(* Logix 5000 project; controller cal1615 1756-L62 rev 20.11; software revision 20.05; part 54 of 81 *)
(* tags used below, declared in another part *)
   FAULT : BOOL;   // Fault AFI
   p01_recipe_active : recipe;   // Active Recipe
   p01r09 : routine;   // System Modes
   p01r09_pb_global_reset : BOOL;   // System Modes PB: Global Fault Reset
   p01r13_line_running : BOOL;   // System Line Start Sequence Line Running
   p02_dint_from_hmi : hmi_dint;
   p02_real_from_hmi : hmi_real;   // MOP HMI Iface Real from HMI
   p23_ao_servo_ds_jog_vel_cmd : REAL;   // Impreg Servo Drive Side Jog Velocity Command [in/sec]
   p23_ao_servo_ds_position_cmd : REAL;   // Impreg Servo Drive Side Position Command
   p23_ao_servo_ds_velocity_cmd : REAL;   // Impreg Servo Drive Side Velocity Command
   p23_ao_servo_ds_zero_offset : REAL;   // Impreg Analog Outputs Drive Side Servo Position Offset
   p23_ao_servo_os_jog_vel_cmd : REAL;   // Impreg Servo Operator Side Jog Velocity Command [in/sec]
   p23_ao_servo_os_position_cmd : REAL;   // Impreg Servo Operator Side Position Command
   p23_ao_servo_os_velocity_cmd : REAL;   // Impreg Servo Operator Side Velocity Command
   p23_di_servo_ds : servo_di;   // Impreg Digital Inputs Servo Drive Side
   p23_di_servo_os : servo_di;   // Impreg Digital Inputs Servo Operator Side
   p23_do_servo_ds : servo_do;   // Impreg Digital Outputs Drive Side Servo
   p23_param_servo_open_position : REAL;
   p23r11 : routine;   // Impreg Servo Operator Side
   p23r11_impreg_gap_os : REAL;
   p23r11_offsets : REAL[100];
   p23r11_pos_offset : REAL;
   p23r11_request_jog_fwd : BOOL;   // Impreg Servo Operator Side Requset Jog Forward
   p23r11_request_jog_rev : BOOL;   // Impreg Servo Operator Side Requset Jog Reverse
   p23r11_selected_position : REAL;
   p23r11_timer_fault : TIMER[4];   // Impreg Servo Drive Side Fault Delay
   p23r11_timer_warning : TIMER[4];   // Impreg Servo Drive Side Warning Delay
   p23r12 : routine;   // Impreg Servo Drive Side
   p23r12_gap_sequence_enabled : BOOL;
   p23r12_impreg_gap_ds : REAL;
   p23r12_offsets : REAL[100];
   p23r12_permissive_jog : BOOL;   // Impreg Servo Drive Side Perimssive Jog
   p23r12_pos_offset : REAL;
   p23r12_request_jog_fwd : BOOL;   // Impreg Servo Drive Side Requset Jog Forward
   p23r12_request_jog_rev : BOOL;   // Impreg Servo Drive Side Requset Jog Reverse
   p23r12_request_position : BOOL;   // Impreg Servo Drive Side Request Position
   p23r12_request_start : BOOL;   // Caoter Servo Drive Side Start Request
   p23r12_request_zero : BOOL;   // Impreg Servo Drive Side Request Zero
   p23r12_selected_position : REAL;
   p23r12_servo_not_ready : BOOL;   // Impreg Servo Drive Side Not Ready
   p23r12_servo_status_ab : BOOL;   // Impreg Servo Drive Side AB Status
   p23r12_servo_status_af : BOOL;   // Impreg Servo Drive Side AF Status
   p23r12_servo_status_bb : BOOL;   // Impreg Servo Drive Side BB Status
   p23r12_step_4_dwell : TIMER;
   p23r12_timer : TIMER[4];   // Impreg Servo Drive Side Timer
   p23r12_timer_fault : TIMER[4];   // Impreg Servo Drive Side Fault Delay
   p23r12_timer_warning : TIMER[4];   // Impreg Servo Drive Side Warning Delay
(* P23_Impreg, continued *)

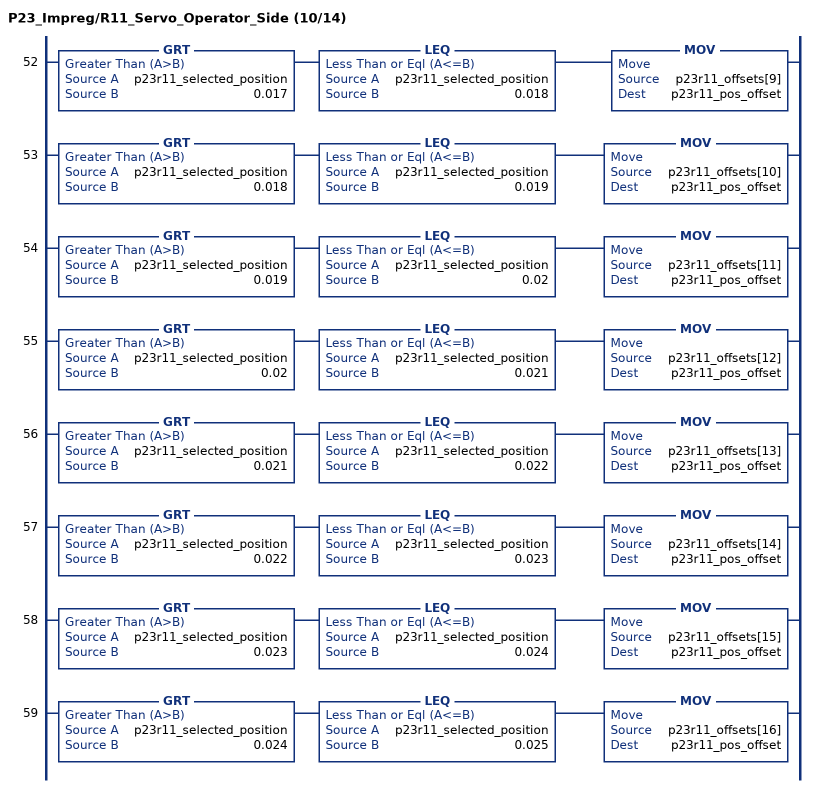
   [picture p1060: P23_Impreg/R11_Servo_Operator_Side rungs 52-59]
   52: GRT(p23r11_selected_position,0.017)LEQ(p23r11_selected_position,0.018)MOV(p23r11_offsets[9],p23r11_pos_offset);
   53: GRT(p23r11_selected_position,0.018)LEQ(p23r11_selected_position,0.019)MOV(p23r11_offsets[10],p23r11_pos_offset);
   54: GRT(p23r11_selected_position,0.019)LEQ(p23r11_selected_position,0.02)MOV(p23r11_offsets[11],p23r11_pos_offset);
   55: GRT(p23r11_selected_position,0.02)LEQ(p23r11_selected_position,0.021)MOV(p23r11_offsets[12],p23r11_pos_offset);
   56: GRT(p23r11_selected_position,0.021)LEQ(p23r11_selected_position,0.022)MOV(p23r11_offsets[13],p23r11_pos_offset);
   57: GRT(p23r11_selected_position,0.022)LEQ(p23r11_selected_position,0.023)MOV(p23r11_offsets[14],p23r11_pos_offset);
   58: GRT(p23r11_selected_position,0.023)LEQ(p23r11_selected_position,0.024)MOV(p23r11_offsets[15],p23r11_pos_offset);
   59: GRT(p23r11_selected_position,0.024)LEQ(p23r11_selected_position,0.025)MOV(p23r11_offsets[16],p23r11_pos_offset);
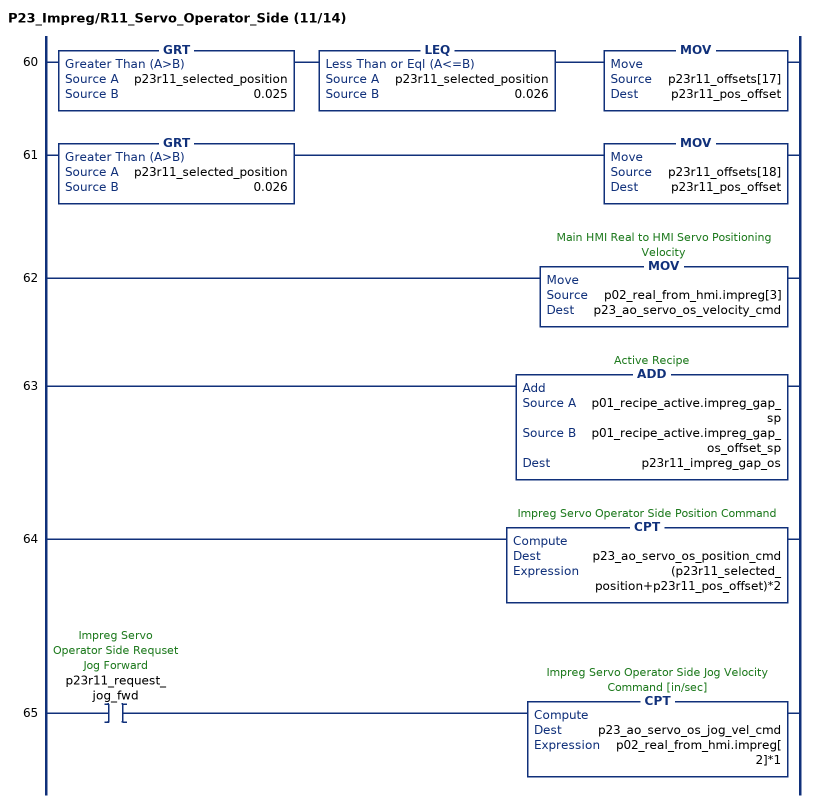
   60: GRT(p23r11_selected_position,0.025)LEQ(p23r11_selected_position,0.026)MOV(p23r11_offsets[17],p23r11_pos_offset);
   61: GRT(p23r11_selected_position,0.026)MOV(p23r11_offsets[18],p23r11_pos_offset);
   62: MOV(p02_real_from_hmi.impreg[3],p23_ao_servo_os_velocity_cmd);
   63: ADD(p01_recipe_active.impreg_gap_sp,p01_recipe_active.impreg_gap_os_offset_sp,p23r11_impreg_gap_os);
   64: CPT(p23_ao_servo_os_position_cmd,(p23r11_selected_position+p23r11_pos_offset)*2);
   65: XIC(p23r11_request_jog_fwd)CPT(p23_ao_servo_os_jog_vel_cmd,p02_real_from_hmi.impreg[2]*1);
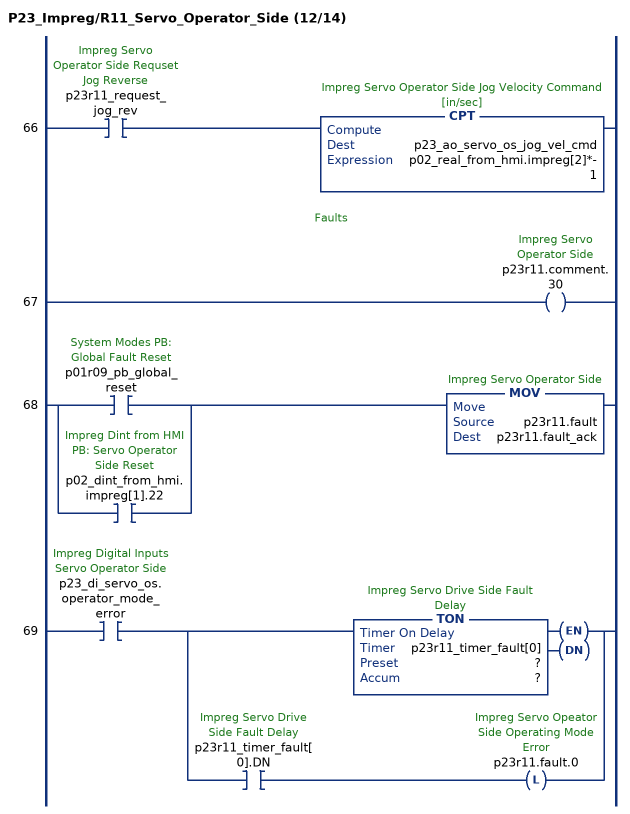
   66: XIC(p23r11_request_jog_rev)CPT(p23_ao_servo_os_jog_vel_cmd,p02_real_from_hmi.impreg[2]*-1);
   // Faults
   67: OTE(p23r11.comment.30);
   68: [XIC(p01r09_pb_global_reset) ,XIC(p02_dint_from_hmi.impreg[1].22) ]MOV(p23r11.fault,p23r11.fault_ack);
   69: XIC(p23_di_servo_os.operator_mode_error)[TON(p23r11_timer_fault[0],?,?) ,XIC(p23r11_timer_fault[0].DN) OTL(p23r11.fault.0) ];
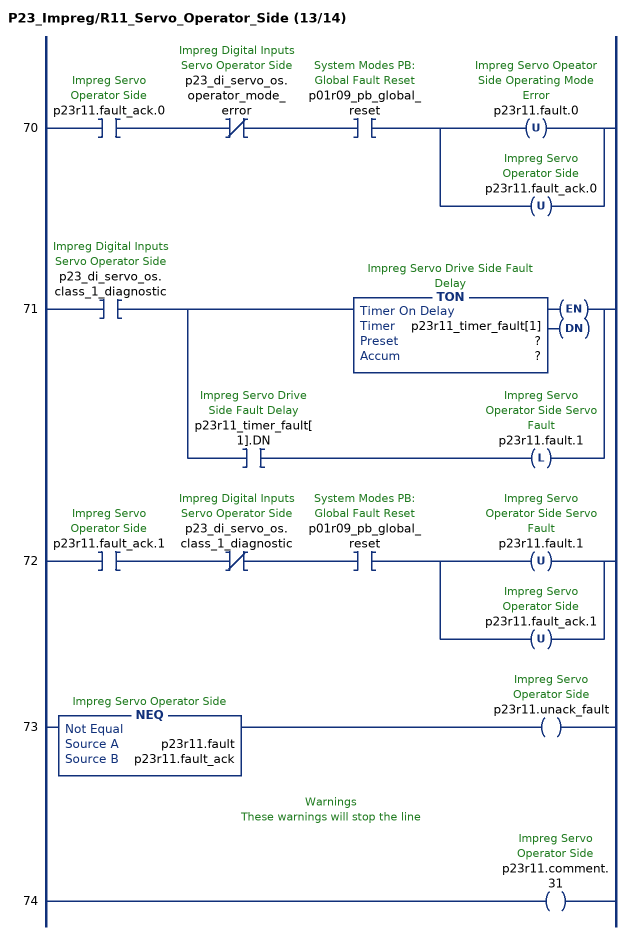
   70: XIC(p23r11.fault_ack.0)XIO(p23_di_servo_os.operator_mode_error)XIC(p01r09_pb_global_reset)[OTU(p23r11.fault.0) ,OTU(p23r11.fault_ack.0) ];
   71: XIC(p23_di_servo_os.class_1_diagnostic)[TON(p23r11_timer_fault[1],?,?) ,XIC(p23r11_timer_fault[1].DN) OTL(p23r11.fault.1) ];
   72: XIC(p23r11.fault_ack.1)XIO(p23_di_servo_os.class_1_diagnostic)XIC(p01r09_pb_global_reset)[OTU(p23r11.fault.1) ,OTU(p23r11.fault_ack.1) ];
   73: NEQ(p23r11.fault,p23r11.fault_ack)OTE(p23r11.unack_fault);
   // Warnings
   // These warnings will stop the line
   74: OTE(p23r11.comment.31);
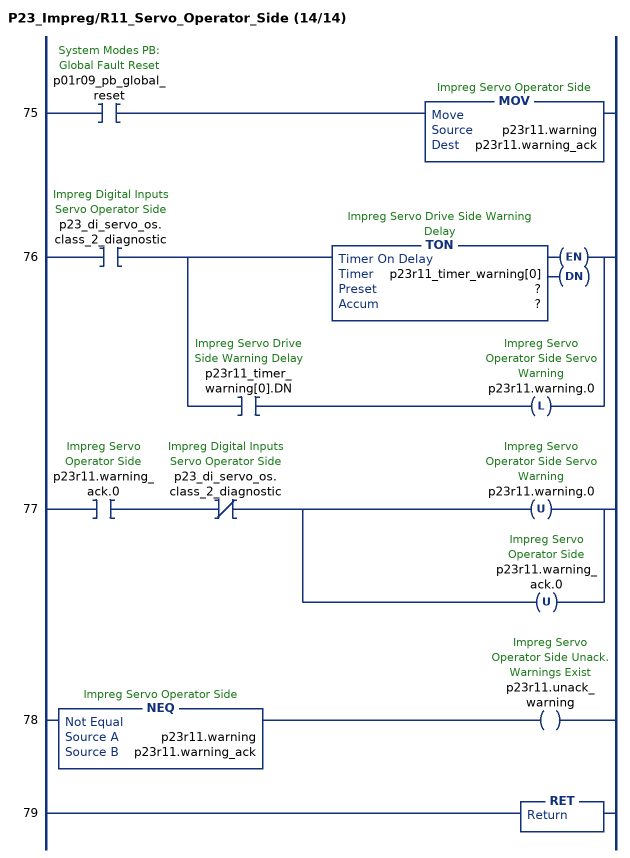
   75: XIC(p01r09_pb_global_reset)MOV(p23r11.warning,p23r11.warning_ack);
   76: XIC(p23_di_servo_os.class_2_diagnostic)[TON(p23r11_timer_warning[0],?,?) ,XIC(p23r11_timer_warning[0].DN) OTL(p23r11.warning.0) ];
   77: XIC(p23r11.warning_ack.0)XIO(p23_di_servo_os.class_2_diagnostic)[OTU(p23r11.warning.0) ,OTU(p23r11.warning_ack.0) ];
   78: NEQ(p23r11.warning,p23r11.warning_ack)OTE(p23r11.unack_warning);
   79: RET();
END_ROUTINE

ROUTINE R12_Servo_Drive_Side   (* ladder *)
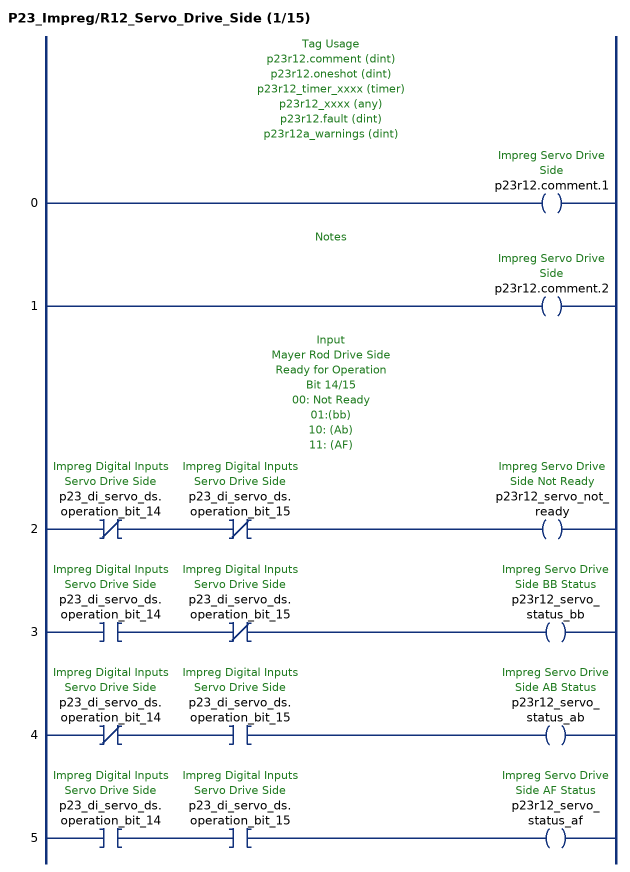
   // Tag Usage
   // p23r12.comment (dint)
   // p23r12.oneshot (dint)
   // p23r12_timer_xxxx (timer)
   // p23r12_xxxx (any)
   // p23r12.fault (dint)
   // p23r12a_warnings (dint)
   0: OTE(p23r12.comment.1);
   // Notes
   1: OTE(p23r12.comment.2);
   // Input
   // Mayer Rod Drive Side
   // Ready for Operation
   // Bit 14/15
   // 00: Not Ready
   // 01:(bb)
   // 10: (Ab)
   // 11: (AF)
   2: XIO(p23_di_servo_ds.operation_bit_14)XIO(p23_di_servo_ds.operation_bit_15)OTE(p23r12_servo_not_ready);
   3: XIC(p23_di_servo_ds.operation_bit_14)XIO(p23_di_servo_ds.operation_bit_15)OTE(p23r12_servo_status_bb);
   4: XIO(p23_di_servo_ds.operation_bit_14)XIC(p23_di_servo_ds.operation_bit_15)OTE(p23r12_servo_status_ab);
   5: XIC(p23_di_servo_ds.operation_bit_14)XIC(p23_di_servo_ds.operation_bit_15)OTE(p23r12_servo_status_af);
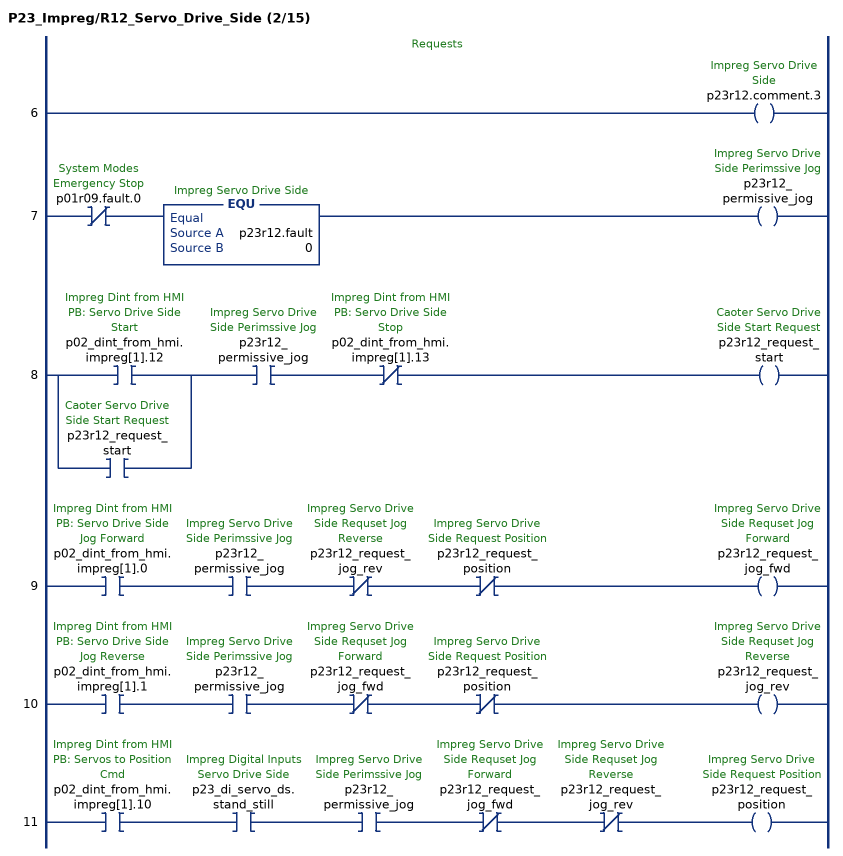
   // Requests
   6: OTE(p23r12.comment.3);
   7: XIO(p01r09.fault.0)EQU(p23r12.fault,0)OTE(p23r12_permissive_jog);
   8: [XIC(p02_dint_from_hmi.impreg[1].12) ,XIC(p23r12_request_start) ]XIC(p23r12_permissive_jog)XIO(p02_dint_from_hmi.impreg[1].13)OTE(p23r12_request_start);
   9: XIC(p02_dint_from_hmi.impreg[1].0)XIC(p23r12_permissive_jog)XIO(p23r12_request_jog_rev)XIO(p23r12_request_position)OTE(p23r12_request_jog_fwd);
   10: XIC(p02_dint_from_hmi.impreg[1].1)XIC(p23r12_permissive_jog)XIO(p23r12_request_jog_fwd)XIO(p23r12_request_position)OTE(p23r12_request_jog_rev);
   11: XIC(p02_dint_from_hmi.impreg[1].10)XIC(p23_di_servo_ds.stand_still)XIC(p23r12_permissive_jog)XIO(p23r12_request_jog_fwd)XIO(p23r12_request_jog_rev)OTE(p23r12_request_position);
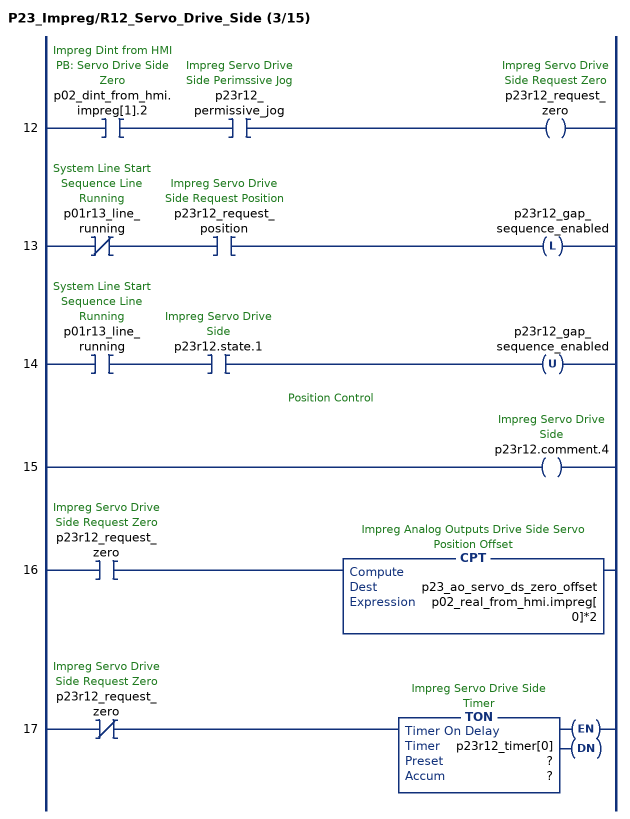
   12: XIC(p02_dint_from_hmi.impreg[1].2)XIC(p23r12_permissive_jog)OTE(p23r12_request_zero);
   13: XIO(p01r13_line_running)XIC(p23r12_request_position)OTL(p23r12_gap_sequence_enabled);
   14: XIC(p01r13_line_running)XIC(p23r12.state.1)OTU(p23r12_gap_sequence_enabled);
   // Position Control
   15: OTE(p23r12.comment.4);
   16: XIC(p23r12_request_zero)CPT(p23_ao_servo_ds_zero_offset,p02_real_from_hmi.impreg[0]*2);
   17: XIO(p23r12_request_zero)TON(p23r12_timer[0],?,?);
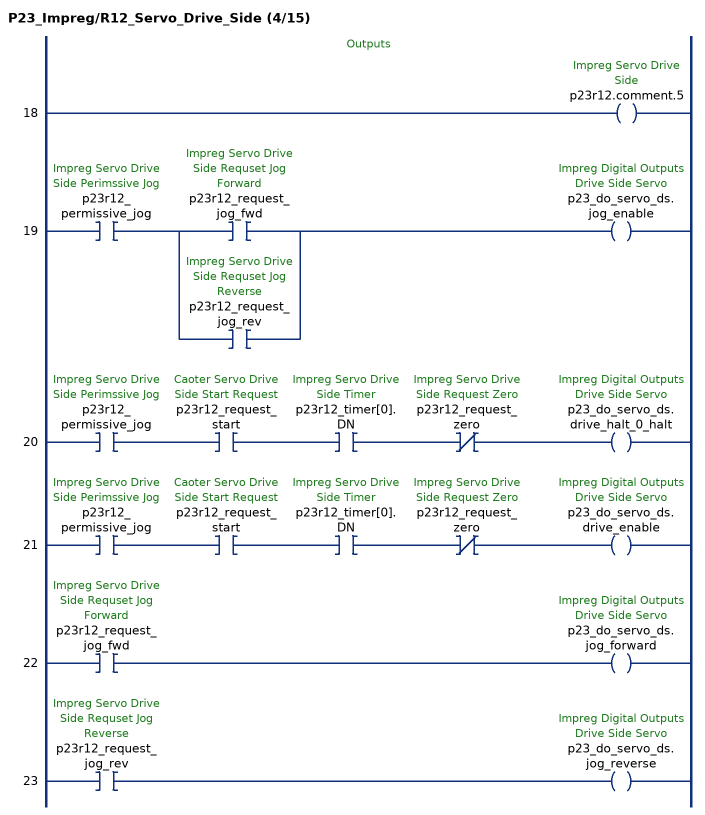
   // Outputs
   18: OTE(p23r12.comment.5);
   19: XIC(p23r12_permissive_jog)[XIC(p23r12_request_jog_fwd) ,XIC(p23r12_request_jog_rev) ]OTE(p23_do_servo_ds.jog_enable);
   20: XIC(p23r12_permissive_jog)XIC(p23r12_request_start)XIC(p23r12_timer[0].DN)XIO(p23r12_request_zero)OTE(p23_do_servo_ds.drive_halt_0_halt);
   21: XIC(p23r12_permissive_jog)XIC(p23r12_request_start)XIC(p23r12_timer[0].DN)XIO(p23r12_request_zero)OTE(p23_do_servo_ds.drive_enable);
   22: XIC(p23r12_request_jog_fwd)OTE(p23_do_servo_ds.jog_forward);
   23: XIC(p23r12_request_jog_rev)OTE(p23_do_servo_ds.jog_reverse);
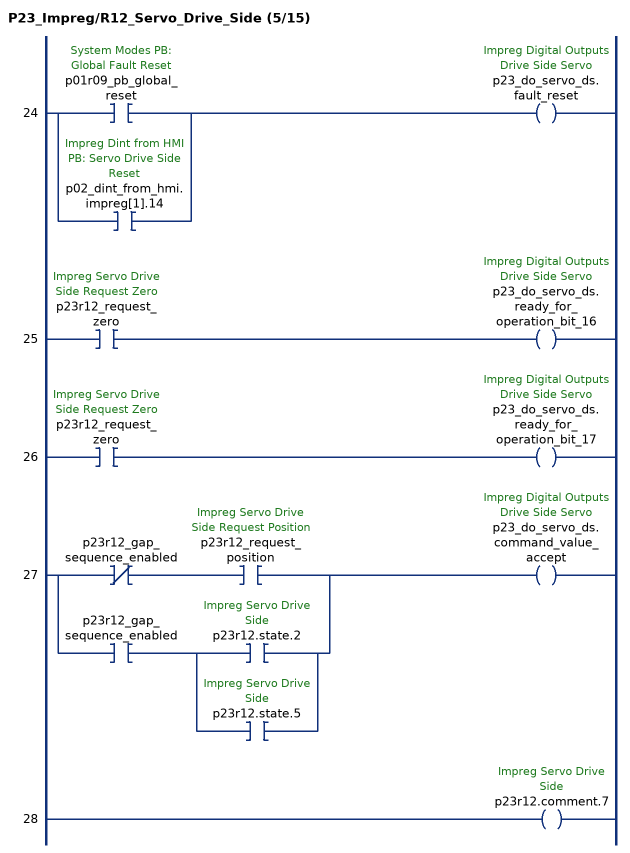
   24: [XIC(p01r09_pb_global_reset) ,XIC(p02_dint_from_hmi.impreg[1].14) ]OTE(p23_do_servo_ds.fault_reset);
   25: XIC(p23r12_request_zero)OTE(p23_do_servo_ds.ready_for_operation_bit_16);
   26: XIC(p23r12_request_zero)OTE(p23_do_servo_ds.ready_for_operation_bit_17);
   27: [XIO(p23r12_gap_sequence_enabled) XIC(p23r12_request_position) ,XIC(p23r12_gap_sequence_enabled) [XIC(p23r12.state.2) ,XIC(p23r12.state.5) ] ]OTE(p23_do_servo_ds.command_value_accept);
   28: OTE(p23r12.comment.7);
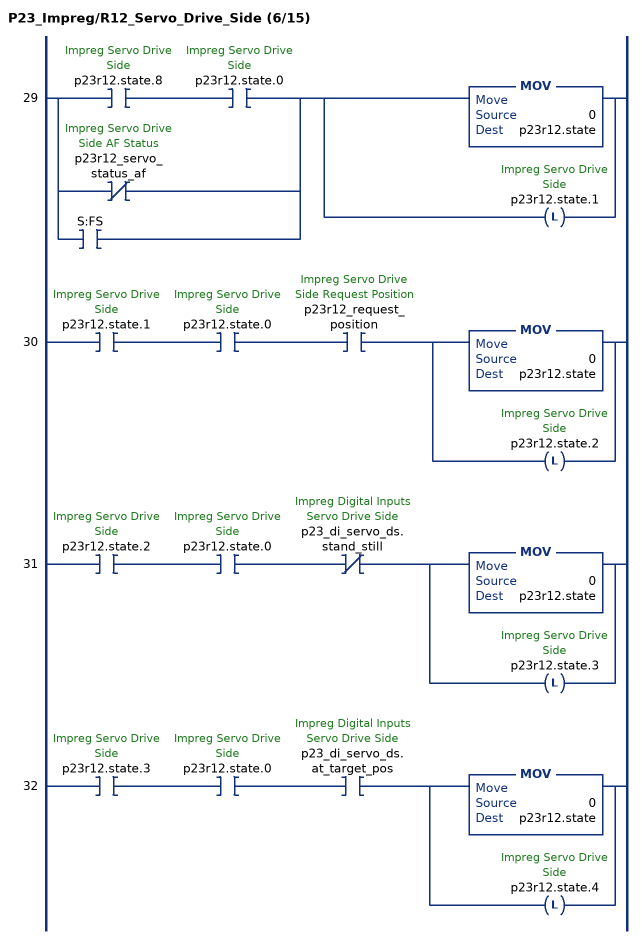
   29: [XIC(p23r12.state.8) XIC(p23r12.state.0) ,XIO(p23r12_servo_status_af) ,XIC(S:FS) ][MOV(0,p23r12.state) ,OTL(p23r12.state.1) ];
   30: XIC(p23r12.state.1)XIC(p23r12.state.0)XIC(p23r12_request_position)[MOV(0,p23r12.state) ,OTL(p23r12.state.2) ];
   31: XIC(p23r12.state.2)XIC(p23r12.state.0)XIO(p23_di_servo_ds.stand_still)[MOV(0,p23r12.state) ,OTL(p23r12.state.3) ];
   32: XIC(p23r12.state.3)XIC(p23r12.state.0)XIC(p23_di_servo_ds.at_target_pos)[MOV(0,p23r12.state) ,OTL(p23r12.state.4) ];
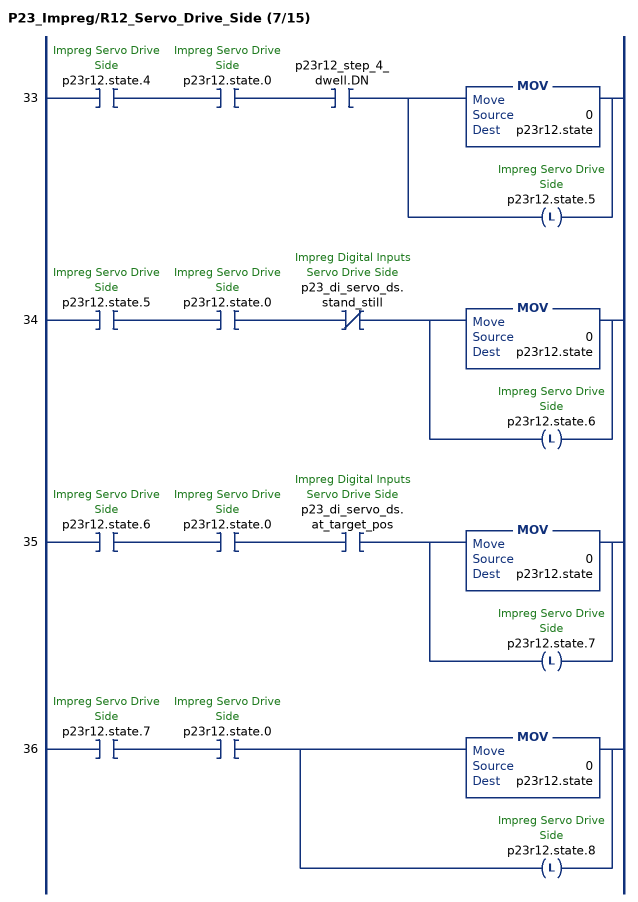
   33: XIC(p23r12.state.4)XIC(p23r12.state.0)XIC(p23r12_step_4_dwell.DN)[MOV(0,p23r12.state) ,OTL(p23r12.state.5) ];
   34: XIC(p23r12.state.5)XIC(p23r12.state.0)XIO(p23_di_servo_ds.stand_still)[MOV(0,p23r12.state) ,OTL(p23r12.state.6) ];
   35: XIC(p23r12.state.6)XIC(p23r12.state.0)XIC(p23_di_servo_ds.at_target_pos)[MOV(0,p23r12.state) ,OTL(p23r12.state.7) ];
   36: XIC(p23r12.state.7)XIC(p23r12.state.0)[MOV(0,p23r12.state) ,OTL(p23r12.state.8) ];
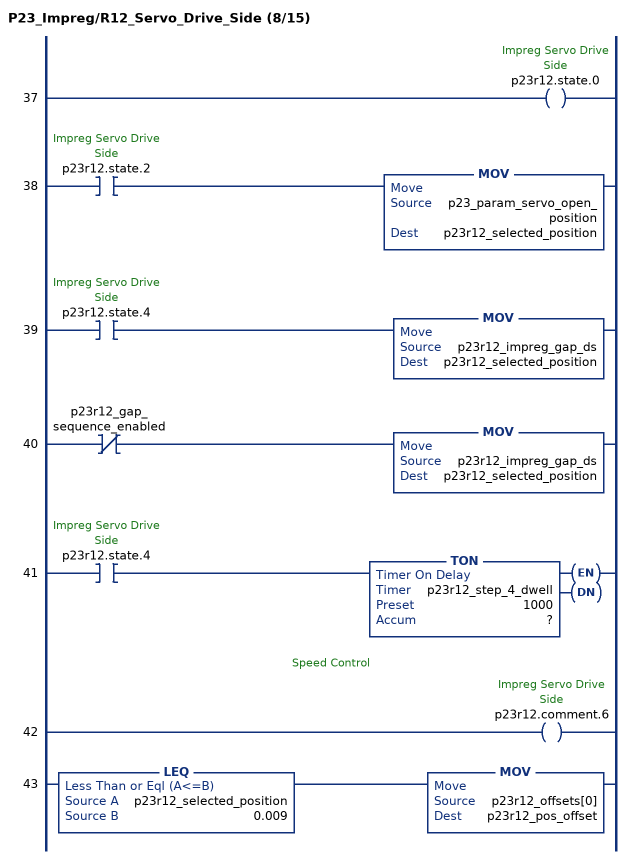
   37: OTE(p23r12.state.0);
   38: XIC(p23r12.state.2)MOV(p23_param_servo_open_position,p23r12_selected_position);
   39: XIC(p23r12.state.4)MOV(p23r12_impreg_gap_ds,p23r12_selected_position);
   40: XIO(p23r12_gap_sequence_enabled)MOV(p23r12_impreg_gap_ds,p23r12_selected_position);
   41: XIC(p23r12.state.4)TON(p23r12_step_4_dwell,?,?);
   // Speed Control
   42: OTE(p23r12.comment.6);
   43: LEQ(p23r12_selected_position,0.009)MOV(p23r12_offsets[0],p23r12_pos_offset);
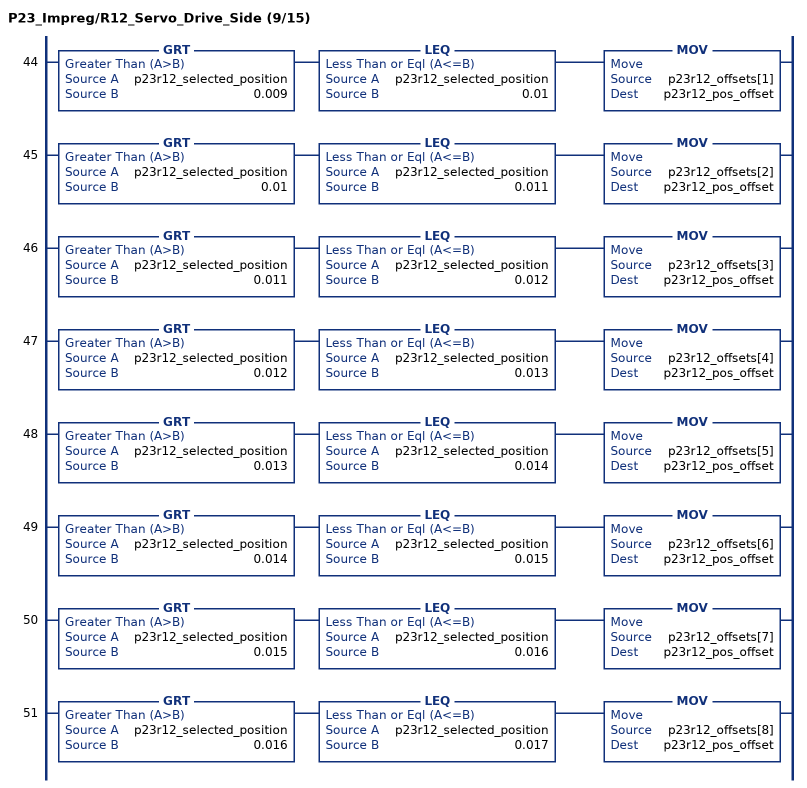
   44: GRT(p23r12_selected_position,0.009)LEQ(p23r12_selected_position,0.01)MOV(p23r12_offsets[1],p23r12_pos_offset);
   45: GRT(p23r12_selected_position,0.01)LEQ(p23r12_selected_position,0.011)MOV(p23r12_offsets[2],p23r12_pos_offset);
   46: GRT(p23r12_selected_position,0.011)LEQ(p23r12_selected_position,0.012)MOV(p23r12_offsets[3],p23r12_pos_offset);
   47: GRT(p23r12_selected_position,0.012)LEQ(p23r12_selected_position,0.013)MOV(p23r12_offsets[4],p23r12_pos_offset);
   48: GRT(p23r12_selected_position,0.013)LEQ(p23r12_selected_position,0.014)MOV(p23r12_offsets[5],p23r12_pos_offset);
   49: GRT(p23r12_selected_position,0.014)LEQ(p23r12_selected_position,0.015)MOV(p23r12_offsets[6],p23r12_pos_offset);
   50: GRT(p23r12_selected_position,0.015)LEQ(p23r12_selected_position,0.016)MOV(p23r12_offsets[7],p23r12_pos_offset);
   51: GRT(p23r12_selected_position,0.016)LEQ(p23r12_selected_position,0.017)MOV(p23r12_offsets[8],p23r12_pos_offset);
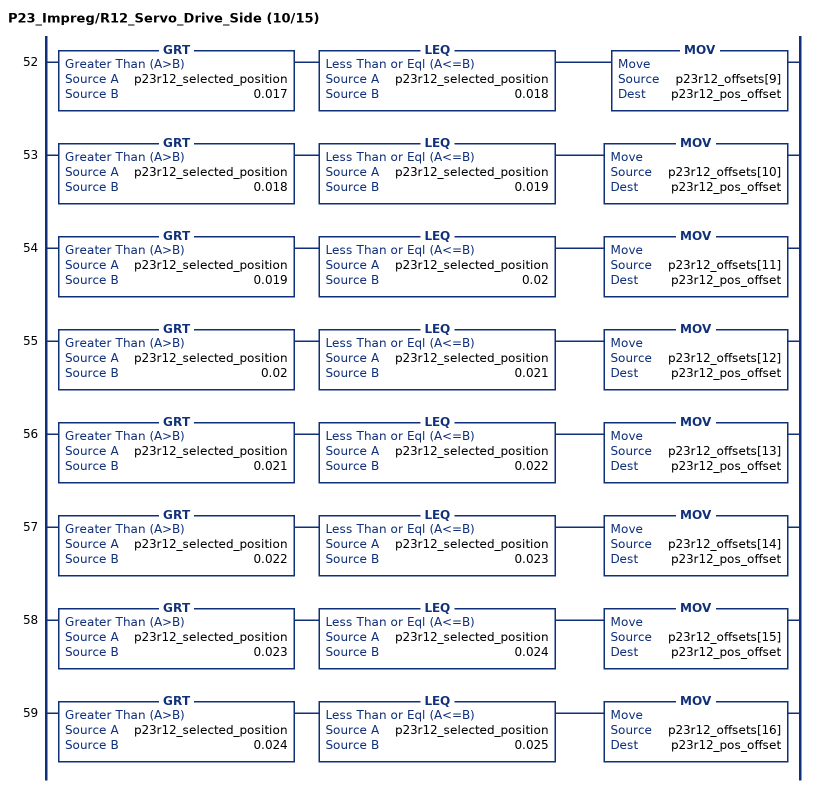
   52: GRT(p23r12_selected_position,0.017)LEQ(p23r12_selected_position,0.018)MOV(p23r12_offsets[9],p23r12_pos_offset);
   53: GRT(p23r12_selected_position,0.018)LEQ(p23r12_selected_position,0.019)MOV(p23r12_offsets[10],p23r12_pos_offset);
   54: GRT(p23r12_selected_position,0.019)LEQ(p23r12_selected_position,0.02)MOV(p23r12_offsets[11],p23r12_pos_offset);
   55: GRT(p23r12_selected_position,0.02)LEQ(p23r12_selected_position,0.021)MOV(p23r12_offsets[12],p23r12_pos_offset);
   56: GRT(p23r12_selected_position,0.021)LEQ(p23r12_selected_position,0.022)MOV(p23r12_offsets[13],p23r12_pos_offset);
   57: GRT(p23r12_selected_position,0.022)LEQ(p23r12_selected_position,0.023)MOV(p23r12_offsets[14],p23r12_pos_offset);
   58: GRT(p23r12_selected_position,0.023)LEQ(p23r12_selected_position,0.024)MOV(p23r12_offsets[15],p23r12_pos_offset);
   59: GRT(p23r12_selected_position,0.024)LEQ(p23r12_selected_position,0.025)MOV(p23r12_offsets[16],p23r12_pos_offset);
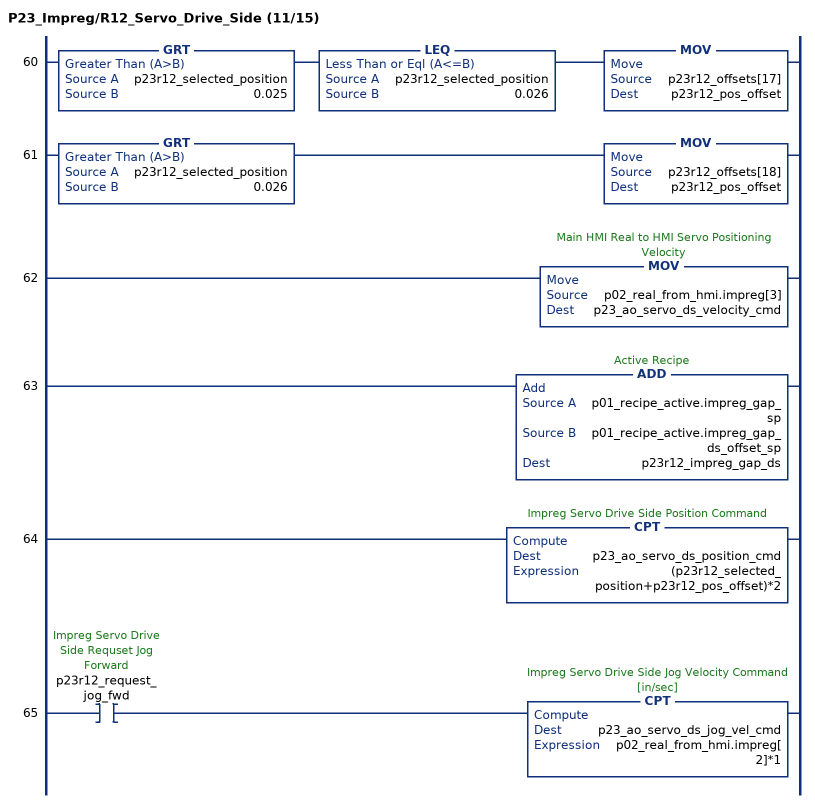
   60: GRT(p23r12_selected_position,0.025)LEQ(p23r12_selected_position,0.026)MOV(p23r12_offsets[17],p23r12_pos_offset);
   61: GRT(p23r12_selected_position,0.026)MOV(p23r12_offsets[18],p23r12_pos_offset);
   62: MOV(p02_real_from_hmi.impreg[3],p23_ao_servo_ds_velocity_cmd);
   63: ADD(p01_recipe_active.impreg_gap_sp,p01_recipe_active.impreg_gap_ds_offset_sp,p23r12_impreg_gap_ds);
   64: CPT(p23_ao_servo_ds_position_cmd,(p23r12_selected_position+p23r12_pos_offset)*2);
   65: XIC(p23r12_request_jog_fwd)CPT(p23_ao_servo_ds_jog_vel_cmd,p02_real_from_hmi.impreg[2]*1);
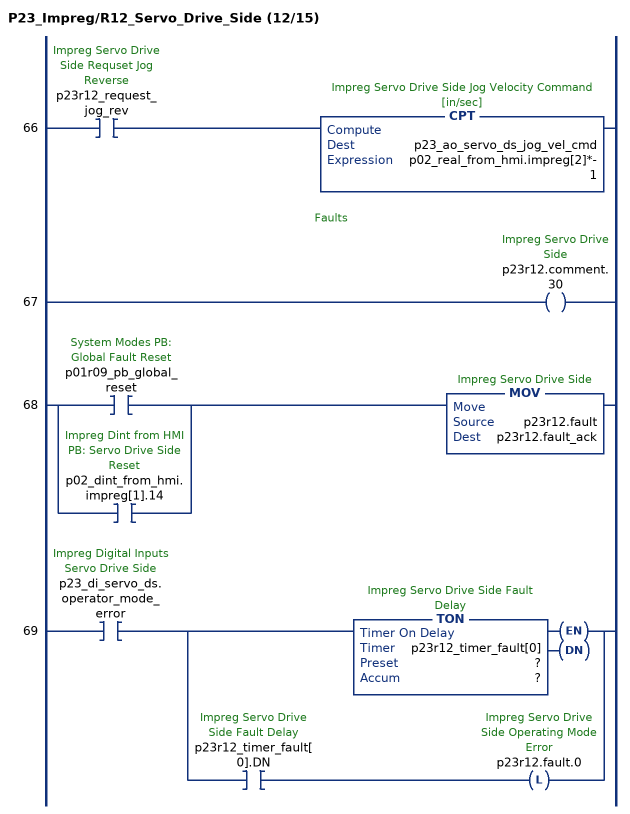
   66: XIC(p23r12_request_jog_rev)CPT(p23_ao_servo_ds_jog_vel_cmd,p02_real_from_hmi.impreg[2]*-1);
   // Faults
   67: OTE(p23r12.comment.30);
   68: [XIC(p01r09_pb_global_reset) ,XIC(p02_dint_from_hmi.impreg[1].14) ]MOV(p23r12.fault,p23r12.fault_ack);
   69: XIC(p23_di_servo_ds.operator_mode_error)[TON(p23r12_timer_fault[0],?,?) ,XIC(p23r12_timer_fault[0].DN) OTL(p23r12.fault.0) ];
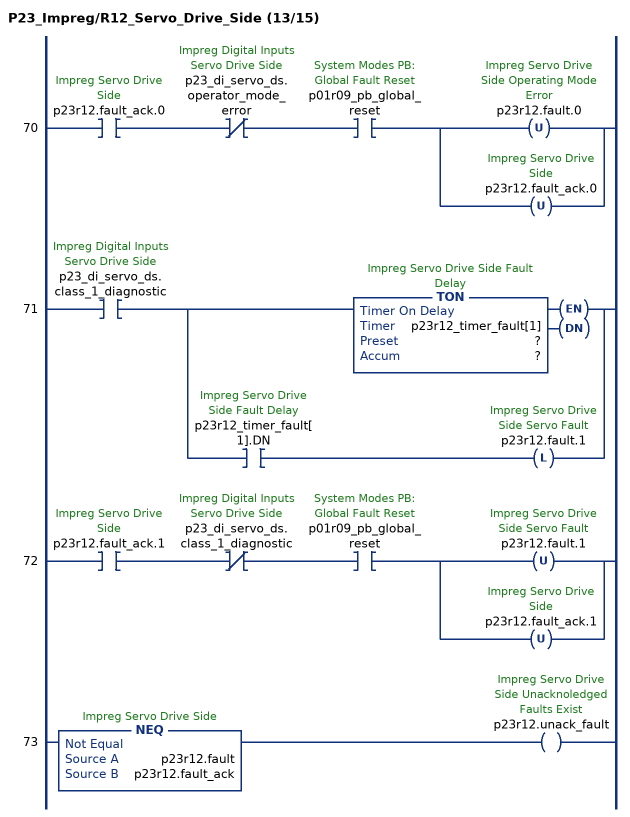
   70: XIC(p23r12.fault_ack.0)XIO(p23_di_servo_ds.operator_mode_error)XIC(p01r09_pb_global_reset)[OTU(p23r12.fault.0) ,OTU(p23r12.fault_ack.0) ];
   71: XIC(p23_di_servo_ds.class_1_diagnostic)[TON(p23r12_timer_fault[1],?,?) ,XIC(p23r12_timer_fault[1].DN) OTL(p23r12.fault.1) ];
   72: XIC(p23r12.fault_ack.1)XIO(p23_di_servo_ds.class_1_diagnostic)XIC(p01r09_pb_global_reset)[OTU(p23r12.fault.1) ,OTU(p23r12.fault_ack.1) ];
   73: NEQ(p23r12.fault,p23r12.fault_ack)OTE(p23r12.unack_fault);
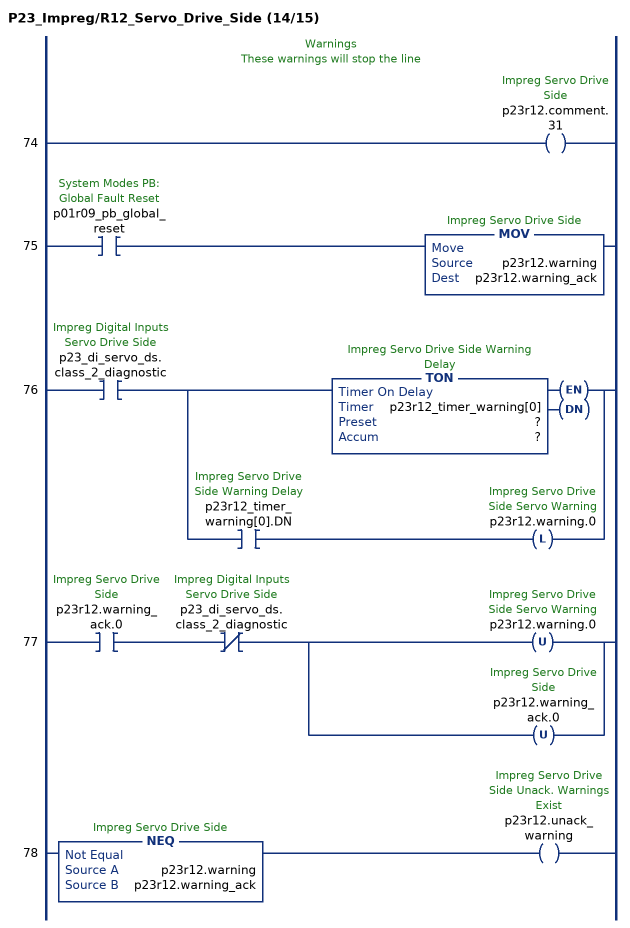
   // Warnings
   // These warnings will stop the line
   74: OTE(p23r12.comment.31);
   75: XIC(p01r09_pb_global_reset)MOV(p23r12.warning,p23r12.warning_ack);
   76: XIC(p23_di_servo_ds.class_2_diagnostic)[TON(p23r12_timer_warning[0],?,?) ,XIC(p23r12_timer_warning[0].DN) OTL(p23r12.warning.0) ];
   77: XIC(p23r12.warning_ack.0)XIO(p23_di_servo_ds.class_2_diagnostic)[OTU(p23r12.warning.0) ,OTU(p23r12.warning_ack.0) ];
   78: NEQ(p23r12.warning,p23r12.warning_ack)OTE(p23r12.unack_warning);
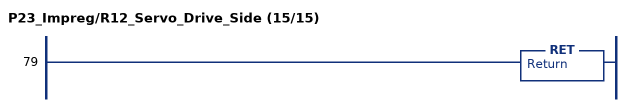
   79: RET();
END_ROUTINE
